REGION Network 108: M611-UNIT 02 FIXTURE 3 TWIN NC UNCLAMP SEQUENCE (TOGGLED) / M100-CLAMP SEQUENCE FIXTURE 1
   RUNG wire#powerrail
      Contact( "DB334_EXTENDED_M_CODE_UNIT_02_STA_0".M_code[611] )
      wire#w1
      I_Contact( "DB334_EXTENDED_M_CODE_UNIT_02_STA_0".M_code[611] )
      wire#w2
      I_Contact( "DB356_M_UNIT_02_STA_0".M_CODES_UNIT_02_STA_0.Ack_M611 )
      I_Contact( "DB2120_MPP_ITC_IPC".RESET_FAULTS )
      I_Contact( "DB356_M_UNIT_02_STA_0".M_CODES_UNIT_02_STA_0.M_RESET_PULSE )
      Coil( "DB356_M_UNIT_02_STA_0".M_CODES_UNIT_02_STA_0.M611 )
   END_RUNG
   RUNG wire#powerrail
      Contact( "DB356_M_UNIT_02_STA_0".M_CODES_UNIT_02_STA_0.M611 )
   END_RUNG wire#w1
   RUNG wire#w1
      I_Contact( "DB356_M_UNIT_02_STA_0".M_CODES_UNIT_02_STA_0.M611 )
   END_RUNG wire#w2
   // the same network as SCL:
   "DB356_M_UNIT_02_STA_0".M_CODES_UNIT_02_STA_0.M611 := ("DB334_EXTENDED_M_CODE_UNIT_02_STA_0".M_code[611] OR "DB356_M_UNIT_02_STA_0".M_CODES_UNIT_02_STA_0.M611) AND (NOT "DB334_EXTENDED_M_CODE_UNIT_02_STA_0".M_code[611] OR NOT "DB356_M_UNIT_02_STA_0".M_CODES_UNIT_02_STA_0.M611) AND NOT "DB356_M_UNIT_02_STA_0".M_CODES_UNIT_02_STA_0.Ack_M611 AND NOT "DB2120_MPP_ITC_IPC".RESET_FAULTS AND NOT "DB356_M_UNIT_02_STA_0".M_CODES_UNIT_02_STA_0.M_RESET_PULSE;
END_REGION

REGION Network 109: ACKNOWLEDGE M620- UNIT 02 FIXTURE 3 GRIPPER CLOSE (READ-IN DISABLE)
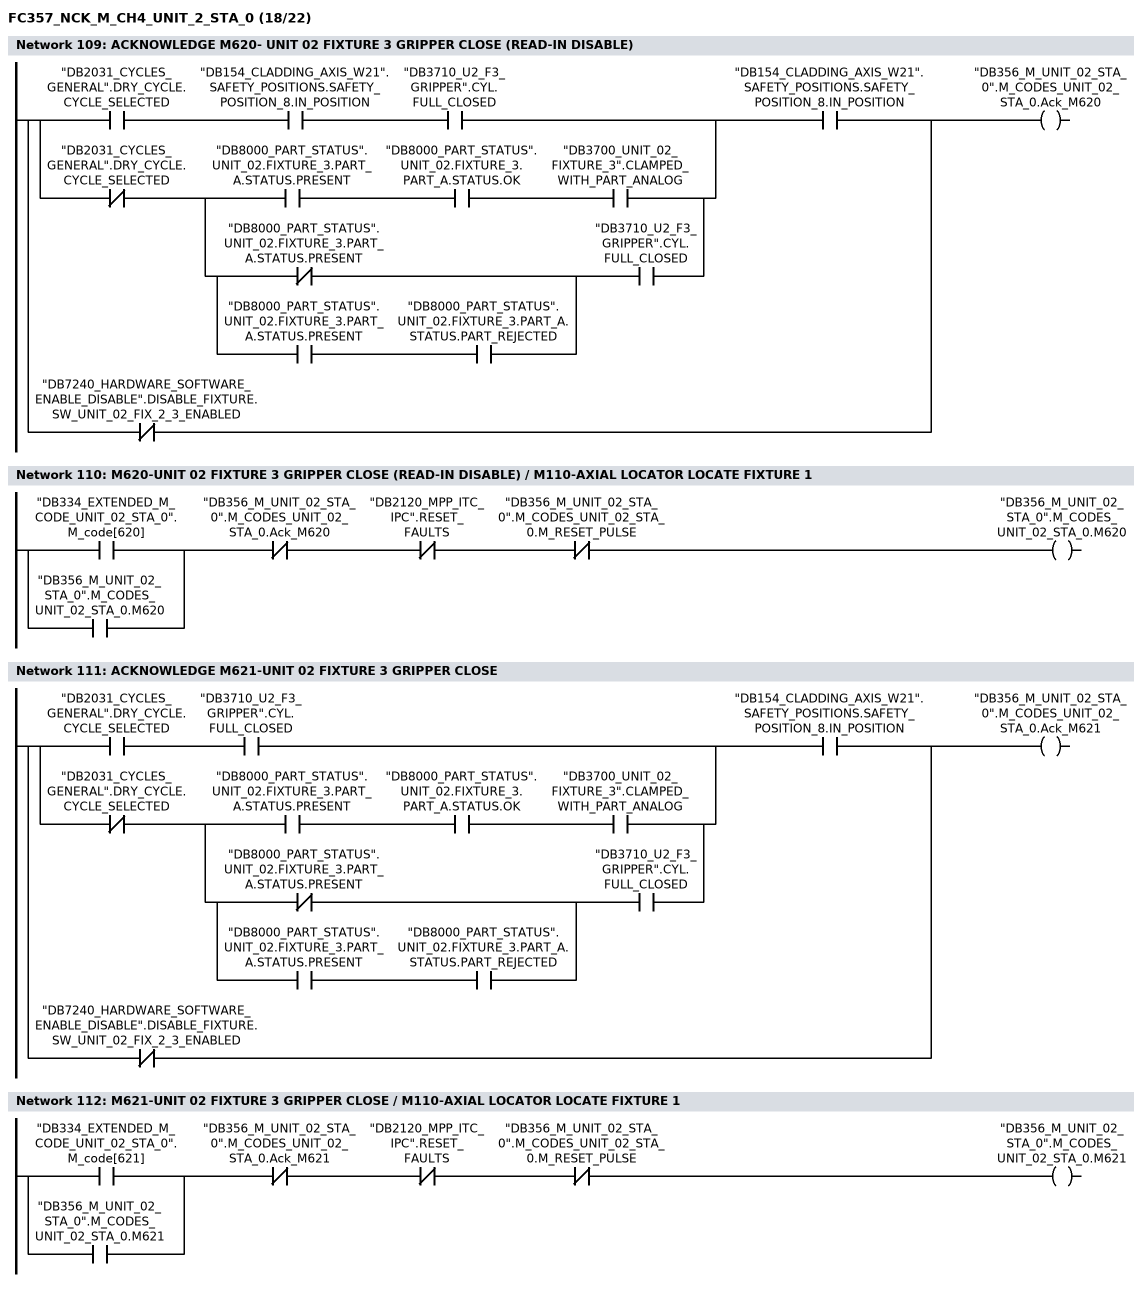
   RUNG wire#powerrail
      Contact( "DB2031_CYCLES_GENERAL".DRY_CYCLE.CYCLE_SELECTED )
      Contact( "DB154_CLADDING_AXIS_W21".SAFETY_POSITIONS.SAFETY_POSITION_8.IN_POSITION )
      Contact( "DB3710_U2_F3_GRIPPER".CYL.FULL_CLOSED )
      wire#w1
      Contact( "DB154_CLADDING_AXIS_W21".SAFETY_POSITIONS.SAFETY_POSITION_8.IN_POSITION )
      wire#w4
      Coil( "DB356_M_UNIT_02_STA_0".M_CODES_UNIT_02_STA_0.Ack_M620 )
   END_RUNG
   RUNG wire#powerrail
      I_Contact( "DB2031_CYCLES_GENERAL".DRY_CYCLE.CYCLE_SELECTED )
      wire#w2
      Contact( "DB8000_PART_STATUS".UNIT_02.FIXTURE_3.PART_A.STATUS.PRESENT )
      Contact( "DB8000_PART_STATUS".UNIT_02.FIXTURE_3.PART_A.STATUS.OK )
      Contact( "DB3700_UNIT_02_FIXTURE_3".CLAMPED_WITH_PART_ANALOG )
   END_RUNG wire#w1
   RUNG wire#w2
      I_Contact( "DB8000_PART_STATUS".UNIT_02.FIXTURE_3.PART_A.STATUS.PRESENT )
      wire#w3
      Contact( "DB3710_U2_F3_GRIPPER".CYL.FULL_CLOSED )
   END_RUNG wire#w1
   RUNG wire#w2
      Contact( "DB8000_PART_STATUS".UNIT_02.FIXTURE_3.PART_A.STATUS.PRESENT )
      Contact( "DB8000_PART_STATUS".UNIT_02.FIXTURE_3.PART_A.STATUS.PART_REJECTED )
   END_RUNG wire#w3
   RUNG wire#powerrail
      I_Contact( "DB7240_HARDWARE_SOFTWARE_ENABLE_DISABLE".DISABLE_FIXTURE.SW_UNIT_02_FIX_2_3_ENABLED )
   END_RUNG wire#w4
   // the same network as SCL:
   "DB356_M_UNIT_02_STA_0".M_CODES_UNIT_02_STA_0.Ack_M620 := ((("DB2031_CYCLES_GENERAL".DRY_CYCLE.CYCLE_SELECTED AND "DB154_CLADDING_AXIS_W21".SAFETY_POSITIONS.SAFETY_POSITION_8.IN_POSITION AND "DB3710_U2_F3_GRIPPER".CYL.FULL_CLOSED) OR (NOT "DB2031_CYCLES_GENERAL".DRY_CYCLE.CYCLE_SELECTED AND (("DB8000_PART_STATUS".UNIT_02.FIXTURE_3.PART_A.STATUS.PRESENT AND "DB8000_PART_STATUS".UNIT_02.FIXTURE_3.PART_A.STATUS.OK AND "DB3700_UNIT_02_FIXTURE_3".CLAMPED_WITH_PART_ANALOG) OR ((NOT "DB8000_PART_STATUS".UNIT_02.FIXTURE_3.PART_A.STATUS.PRESENT OR ("DB8000_PART_STATUS".UNIT_02.FIXTURE_3.PART_A.STATUS.PRESENT AND "DB8000_PART_STATUS".UNIT_02.FIXTURE_3.PART_A.STATUS.PART_REJECTED)) AND "DB3710_U2_F3_GRIPPER".CYL.FULL_CLOSED)))) AND "DB154_CLADDING_AXIS_W21".SAFETY_POSITIONS.SAFETY_POSITION_8.IN_POSITION) OR NOT "DB7240_HARDWARE_SOFTWARE_ENABLE_DISABLE".DISABLE_FIXTURE.SW_UNIT_02_FIX_2_3_ENABLED;
END_REGION

REGION Network 110: M620-UNIT 02 FIXTURE 3 GRIPPER CLOSE (READ-IN DISABLE) / M110-AXIAL LOCATOR LOCATE FIXTURE 1
   RUNG wire#powerrail
      Contact( "DB334_EXTENDED_M_CODE_UNIT_02_STA_0".M_code[620] )
      wire#w1
      I_Contact( "DB356_M_UNIT_02_STA_0".M_CODES_UNIT_02_STA_0.Ack_M620 )
      I_Contact( "DB2120_MPP_ITC_IPC".RESET_FAULTS )
      I_Contact( "DB356_M_UNIT_02_STA_0".M_CODES_UNIT_02_STA_0.M_RESET_PULSE )
      Coil( "DB356_M_UNIT_02_STA_0".M_CODES_UNIT_02_STA_0.M620 )
   END_RUNG
   RUNG wire#powerrail
      Contact( "DB356_M_UNIT_02_STA_0".M_CODES_UNIT_02_STA_0.M620 )
   END_RUNG wire#w1
   // the same network as SCL:
   "DB356_M_UNIT_02_STA_0".M_CODES_UNIT_02_STA_0.M620 := ("DB334_EXTENDED_M_CODE_UNIT_02_STA_0".M_code[620] OR "DB356_M_UNIT_02_STA_0".M_CODES_UNIT_02_STA_0.M620) AND NOT "DB356_M_UNIT_02_STA_0".M_CODES_UNIT_02_STA_0.Ack_M620 AND NOT "DB2120_MPP_ITC_IPC".RESET_FAULTS AND NOT "DB356_M_UNIT_02_STA_0".M_CODES_UNIT_02_STA_0.M_RESET_PULSE;
END_REGION

REGION Network 111: ACKNOWLEDGE M621-UNIT 02 FIXTURE 3 GRIPPER CLOSE
   RUNG wire#powerrail
      Contact( "DB2031_CYCLES_GENERAL".DRY_CYCLE.CYCLE_SELECTED )
      Contact( "DB3710_U2_F3_GRIPPER".CYL.FULL_CLOSED )
      wire#w1
      Contact( "DB154_CLADDING_AXIS_W21".SAFETY_POSITIONS.SAFETY_POSITION_8.IN_POSITION )
      wire#w4
      Coil( "DB356_M_UNIT_02_STA_0".M_CODES_UNIT_02_STA_0.Ack_M621 )
   END_RUNG
   RUNG wire#powerrail
      I_Contact( "DB2031_CYCLES_GENERAL".DRY_CYCLE.CYCLE_SELECTED )
      wire#w2
      Contact( "DB8000_PART_STATUS".UNIT_02.FIXTURE_3.PART_A.STATUS.PRESENT )
      Contact( "DB8000_PART_STATUS".UNIT_02.FIXTURE_3.PART_A.STATUS.OK )
      Contact( "DB3700_UNIT_02_FIXTURE_3".CLAMPED_WITH_PART_ANALOG )
   END_RUNG wire#w1
   RUNG wire#w2
      I_Contact( "DB8000_PART_STATUS".UNIT_02.FIXTURE_3.PART_A.STATUS.PRESENT )
      wire#w3
      Contact( "DB3710_U2_F3_GRIPPER".CYL.FULL_CLOSED )
   END_RUNG wire#w1
   RUNG wire#w2
      Contact( "DB8000_PART_STATUS".UNIT_02.FIXTURE_3.PART_A.STATUS.PRESENT )
      Contact( "DB8000_PART_STATUS".UNIT_02.FIXTURE_3.PART_A.STATUS.PART_REJECTED )
   END_RUNG wire#w3
   RUNG wire#powerrail
      I_Contact( "DB7240_HARDWARE_SOFTWARE_ENABLE_DISABLE".DISABLE_FIXTURE.SW_UNIT_02_FIX_2_3_ENABLED )
   END_RUNG wire#w4
   // the same network as SCL:
   "DB356_M_UNIT_02_STA_0".M_CODES_UNIT_02_STA_0.Ack_M621 := ((("DB2031_CYCLES_GENERAL".DRY_CYCLE.CYCLE_SELECTED AND "DB3710_U2_F3_GRIPPER".CYL.FULL_CLOSED) OR (NOT "DB2031_CYCLES_GENERAL".DRY_CYCLE.CYCLE_SELECTED AND (("DB8000_PART_STATUS".UNIT_02.FIXTURE_3.PART_A.STATUS.PRESENT AND "DB8000_PART_STATUS".UNIT_02.FIXTURE_3.PART_A.STATUS.OK AND "DB3700_UNIT_02_FIXTURE_3".CLAMPED_WITH_PART_ANALOG) OR ((NOT "DB8000_PART_STATUS".UNIT_02.FIXTURE_3.PART_A.STATUS.PRESENT OR ("DB8000_PART_STATUS".UNIT_02.FIXTURE_3.PART_A.STATUS.PRESENT AND "DB8000_PART_STATUS".UNIT_02.FIXTURE_3.PART_A.STATUS.PART_REJECTED)) AND "DB3710_U2_F3_GRIPPER".CYL.FULL_CLOSED)))) AND "DB154_CLADDING_AXIS_W21".SAFETY_POSITIONS.SAFETY_POSITION_8.IN_POSITION) OR NOT "DB7240_HARDWARE_SOFTWARE_ENABLE_DISABLE".DISABLE_FIXTURE.SW_UNIT_02_FIX_2_3_ENABLED;
END_REGION

REGION Network 112: M621-UNIT 02 FIXTURE 3 GRIPPER CLOSE / M110-AXIAL LOCATOR LOCATE FIXTURE 1
   RUNG wire#powerrail
      Contact( "DB334_EXTENDED_M_CODE_UNIT_02_STA_0".M_code[621] )
      wire#w1
      I_Contact( "DB356_M_UNIT_02_STA_0".M_CODES_UNIT_02_STA_0.Ack_M621 )
      I_Contact( "DB2120_MPP_ITC_IPC".RESET_FAULTS )
      I_Contact( "DB356_M_UNIT_02_STA_0".M_CODES_UNIT_02_STA_0.M_RESET_PULSE )
      Coil( "DB356_M_UNIT_02_STA_0".M_CODES_UNIT_02_STA_0.M621 )
   END_RUNG
   RUNG wire#powerrail
      Contact( "DB356_M_UNIT_02_STA_0".M_CODES_UNIT_02_STA_0.M621 )
   END_RUNG wire#w1
   // the same network as SCL:
   "DB356_M_UNIT_02_STA_0".M_CODES_UNIT_02_STA_0.M621 := ("DB334_EXTENDED_M_CODE_UNIT_02_STA_0".M_code[621] OR "DB356_M_UNIT_02_STA_0".M_CODES_UNIT_02_STA_0.M621) AND NOT "DB356_M_UNIT_02_STA_0".M_CODES_UNIT_02_STA_0.Ack_M621 AND NOT "DB2120_MPP_ITC_IPC".RESET_FAULTS AND NOT "DB356_M_UNIT_02_STA_0".M_CODES_UNIT_02_STA_0.M_RESET_PULSE;
END_REGION

REGION Network 113: ACKNOWLEDGE M622-UNIT 02 FIXTURE 3 GRIPPER OPEN (READ-IN DISABLE) / ACKNOWLEDGE M111-AXIAL LOCATOR RETURN FIXTURE 1
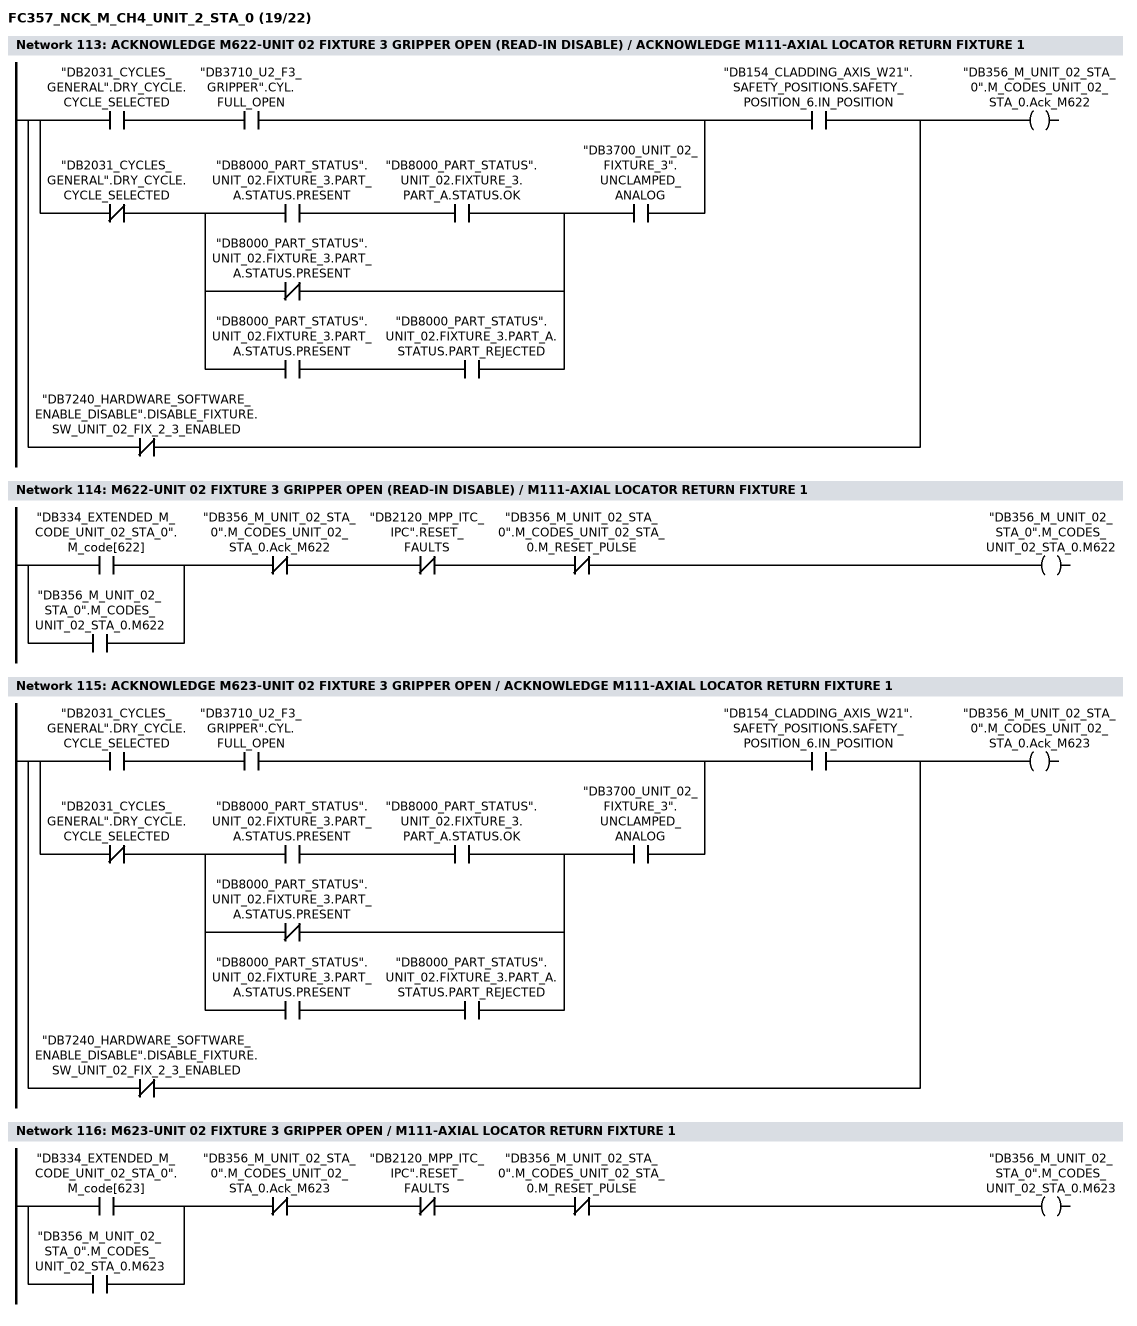
   RUNG wire#powerrail
      Contact( "DB2031_CYCLES_GENERAL".DRY_CYCLE.CYCLE_SELECTED )
      Contact( "DB3710_U2_F3_GRIPPER".CYL.FULL_OPEN )
      wire#w1
      Contact( "DB154_CLADDING_AXIS_W21".SAFETY_POSITIONS.SAFETY_POSITION_6.IN_POSITION )
      wire#w4
      Coil( "DB356_M_UNIT_02_STA_0".M_CODES_UNIT_02_STA_0.Ack_M622 )
   END_RUNG
   RUNG wire#powerrail
      I_Contact( "DB2031_CYCLES_GENERAL".DRY_CYCLE.CYCLE_SELECTED )
      wire#w2
      Contact( "DB8000_PART_STATUS".UNIT_02.FIXTURE_3.PART_A.STATUS.PRESENT )
      Contact( "DB8000_PART_STATUS".UNIT_02.FIXTURE_3.PART_A.STATUS.OK )
      wire#w3
      Contact( "DB3700_UNIT_02_FIXTURE_3".UNCLAMPED_ANALOG )
   END_RUNG wire#w1
   RUNG wire#w2
      I_Contact( "DB8000_PART_STATUS".UNIT_02.FIXTURE_3.PART_A.STATUS.PRESENT )
   END_RUNG wire#w3
   RUNG wire#w2
      Contact( "DB8000_PART_STATUS".UNIT_02.FIXTURE_3.PART_A.STATUS.PRESENT )
      Contact( "DB8000_PART_STATUS".UNIT_02.FIXTURE_3.PART_A.STATUS.PART_REJECTED )
   END_RUNG wire#w3
   RUNG wire#powerrail
      I_Contact( "DB7240_HARDWARE_SOFTWARE_ENABLE_DISABLE".DISABLE_FIXTURE.SW_UNIT_02_FIX_2_3_ENABLED )
   END_RUNG wire#w4
   // the same network as SCL:
   "DB356_M_UNIT_02_STA_0".M_CODES_UNIT_02_STA_0.Ack_M622 := ((("DB2031_CYCLES_GENERAL".DRY_CYCLE.CYCLE_SELECTED AND "DB3710_U2_F3_GRIPPER".CYL.FULL_OPEN) OR (NOT "DB2031_CYCLES_GENERAL".DRY_CYCLE.CYCLE_SELECTED AND (("DB8000_PART_STATUS".UNIT_02.FIXTURE_3.PART_A.STATUS.PRESENT AND "DB8000_PART_STATUS".UNIT_02.FIXTURE_3.PART_A.STATUS.OK) OR NOT "DB8000_PART_STATUS".UNIT_02.FIXTURE_3.PART_A.STATUS.PRESENT OR ("DB8000_PART_STATUS".UNIT_02.FIXTURE_3.PART_A.STATUS.PRESENT AND "DB8000_PART_STATUS".UNIT_02.FIXTURE_3.PART_A.STATUS.PART_REJECTED)) AND "DB3700_UNIT_02_FIXTURE_3".UNCLAMPED_ANALOG)) AND "DB154_CLADDING_AXIS_W21".SAFETY_POSITIONS.SAFETY_POSITION_6.IN_POSITION) OR NOT "DB7240_HARDWARE_SOFTWARE_ENABLE_DISABLE".DISABLE_FIXTURE.SW_UNIT_02_FIX_2_3_ENABLED;
END_REGION

REGION Network 114: M622-UNIT 02 FIXTURE 3 GRIPPER OPEN (READ-IN DISABLE) / M111-AXIAL LOCATOR RETURN FIXTURE 1
   RUNG wire#powerrail
      Contact( "DB334_EXTENDED_M_CODE_UNIT_02_STA_0".M_code[622] )
      wire#w1
      I_Contact( "DB356_M_UNIT_02_STA_0".M_CODES_UNIT_02_STA_0.Ack_M622 )
      I_Contact( "DB2120_MPP_ITC_IPC".RESET_FAULTS )
      I_Contact( "DB356_M_UNIT_02_STA_0".M_CODES_UNIT_02_STA_0.M_RESET_PULSE )
      Coil( "DB356_M_UNIT_02_STA_0".M_CODES_UNIT_02_STA_0.M622 )
   END_RUNG
   RUNG wire#powerrail
      Contact( "DB356_M_UNIT_02_STA_0".M_CODES_UNIT_02_STA_0.M622 )
   END_RUNG wire#w1
   // the same network as SCL:
   "DB356_M_UNIT_02_STA_0".M_CODES_UNIT_02_STA_0.M622 := ("DB334_EXTENDED_M_CODE_UNIT_02_STA_0".M_code[622] OR "DB356_M_UNIT_02_STA_0".M_CODES_UNIT_02_STA_0.M622) AND NOT "DB356_M_UNIT_02_STA_0".M_CODES_UNIT_02_STA_0.Ack_M622 AND NOT "DB2120_MPP_ITC_IPC".RESET_FAULTS AND NOT "DB356_M_UNIT_02_STA_0".M_CODES_UNIT_02_STA_0.M_RESET_PULSE;
END_REGION

REGION Network 115: ACKNOWLEDGE M623-UNIT 02 FIXTURE 3 GRIPPER OPEN / ACKNOWLEDGE M111-AXIAL LOCATOR RETURN FIXTURE 1
   RUNG wire#powerrail
      Contact( "DB2031_CYCLES_GENERAL".DRY_CYCLE.CYCLE_SELECTED )
      Contact( "DB3710_U2_F3_GRIPPER".CYL.FULL_OPEN )
      wire#w1
      Contact( "DB154_CLADDING_AXIS_W21".SAFETY_POSITIONS.SAFETY_POSITION_6.IN_POSITION )
      wire#w4
      Coil( "DB356_M_UNIT_02_STA_0".M_CODES_UNIT_02_STA_0.Ack_M623 )
   END_RUNG
   RUNG wire#powerrail
      I_Contact( "DB2031_CYCLES_GENERAL".DRY_CYCLE.CYCLE_SELECTED )
      wire#w2
      Contact( "DB8000_PART_STATUS".UNIT_02.FIXTURE_3.PART_A.STATUS.PRESENT )
      Contact( "DB8000_PART_STATUS".UNIT_02.FIXTURE_3.PART_A.STATUS.OK )
      wire#w3
      Contact( "DB3700_UNIT_02_FIXTURE_3".UNCLAMPED_ANALOG )
   END_RUNG wire#w1
   RUNG wire#w2
      I_Contact( "DB8000_PART_STATUS".UNIT_02.FIXTURE_3.PART_A.STATUS.PRESENT )
   END_RUNG wire#w3
   RUNG wire#w2
      Contact( "DB8000_PART_STATUS".UNIT_02.FIXTURE_3.PART_A.STATUS.PRESENT )
      Contact( "DB8000_PART_STATUS".UNIT_02.FIXTURE_3.PART_A.STATUS.PART_REJECTED )
   END_RUNG wire#w3
   RUNG wire#powerrail
      I_Contact( "DB7240_HARDWARE_SOFTWARE_ENABLE_DISABLE".DISABLE_FIXTURE.SW_UNIT_02_FIX_2_3_ENABLED )
   END_RUNG wire#w4
   // the same network as SCL:
   "DB356_M_UNIT_02_STA_0".M_CODES_UNIT_02_STA_0.Ack_M623 := ((("DB2031_CYCLES_GENERAL".DRY_CYCLE.CYCLE_SELECTED AND "DB3710_U2_F3_GRIPPER".CYL.FULL_OPEN) OR (NOT "DB2031_CYCLES_GENERAL".DRY_CYCLE.CYCLE_SELECTED AND (("DB8000_PART_STATUS".UNIT_02.FIXTURE_3.PART_A.STATUS.PRESENT AND "DB8000_PART_STATUS".UNIT_02.FIXTURE_3.PART_A.STATUS.OK) OR NOT "DB8000_PART_STATUS".UNIT_02.FIXTURE_3.PART_A.STATUS.PRESENT OR ("DB8000_PART_STATUS".UNIT_02.FIXTURE_3.PART_A.STATUS.PRESENT AND "DB8000_PART_STATUS".UNIT_02.FIXTURE_3.PART_A.STATUS.PART_REJECTED)) AND "DB3700_UNIT_02_FIXTURE_3".UNCLAMPED_ANALOG)) AND "DB154_CLADDING_AXIS_W21".SAFETY_POSITIONS.SAFETY_POSITION_6.IN_POSITION) OR NOT "DB7240_HARDWARE_SOFTWARE_ENABLE_DISABLE".DISABLE_FIXTURE.SW_UNIT_02_FIX_2_3_ENABLED;
END_REGION

REGION Network 116: M623-UNIT 02 FIXTURE 3 GRIPPER OPEN / M111-AXIAL LOCATOR RETURN FIXTURE 1
   RUNG wire#powerrail
      Contact( "DB334_EXTENDED_M_CODE_UNIT_02_STA_0".M_code[623] )
      wire#w1
      I_Contact( "DB356_M_UNIT_02_STA_0".M_CODES_UNIT_02_STA_0.Ack_M623 )
      I_Contact( "DB2120_MPP_ITC_IPC".RESET_FAULTS )
      I_Contact( "DB356_M_UNIT_02_STA_0".M_CODES_UNIT_02_STA_0.M_RESET_PULSE )
      Coil( "DB356_M_UNIT_02_STA_0".M_CODES_UNIT_02_STA_0.M623 )
   END_RUNG
   RUNG wire#powerrail
      Contact( "DB356_M_UNIT_02_STA_0".M_CODES_UNIT_02_STA_0.M623 )
   END_RUNG wire#w1
   // the same network as SCL:
   "DB356_M_UNIT_02_STA_0".M_CODES_UNIT_02_STA_0.M623 := ("DB334_EXTENDED_M_CODE_UNIT_02_STA_0".M_code[623] OR "DB356_M_UNIT_02_STA_0".M_CODES_UNIT_02_STA_0.M623) AND NOT "DB356_M_UNIT_02_STA_0".M_CODES_UNIT_02_STA_0.Ack_M623 AND NOT "DB2120_MPP_ITC_IPC".RESET_FAULTS AND NOT "DB356_M_UNIT_02_STA_0".M_CODES_UNIT_02_STA_0.M_RESET_PULSE;
END_REGION

REGION Network 117: ACKNOWLEDGE M624-UNIT 02 FIXTURE 3 GRIPPER RELEASE PRESSURE (READ-IN DISABLE) / ACKNOWLEDGE M112-AXIAL LOCATOR RELAX FIXTURE 1
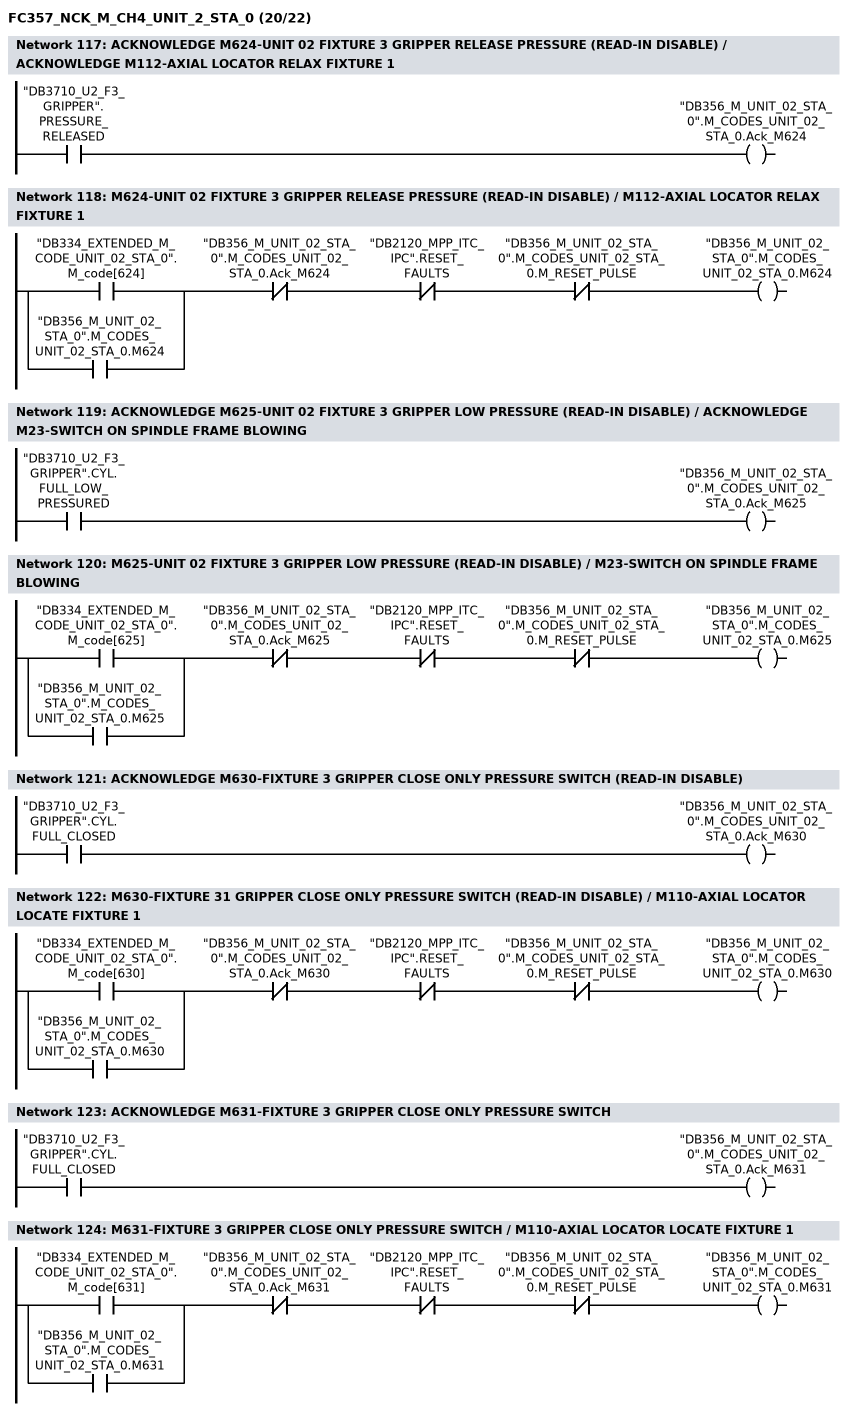
   RUNG wire#powerrail
      Contact( "DB3710_U2_F3_GRIPPER".PRESSURE_RELEASED )
      Coil( "DB356_M_UNIT_02_STA_0".M_CODES_UNIT_02_STA_0.Ack_M624 )
   END_RUNG
   // the same network as SCL:
   "DB356_M_UNIT_02_STA_0".M_CODES_UNIT_02_STA_0.Ack_M624 := "DB3710_U2_F3_GRIPPER".PRESSURE_RELEASED;
END_REGION

REGION Network 118: M624-UNIT 02 FIXTURE 3 GRIPPER RELEASE PRESSURE (READ-IN DISABLE) / M112-AXIAL LOCATOR RELAX FIXTURE 1
   RUNG wire#powerrail
      Contact( "DB334_EXTENDED_M_CODE_UNIT_02_STA_0".M_code[624] )
      wire#w1
      I_Contact( "DB356_M_UNIT_02_STA_0".M_CODES_UNIT_02_STA_0.Ack_M624 )
      I_Contact( "DB2120_MPP_ITC_IPC".RESET_FAULTS )
      I_Contact( "DB356_M_UNIT_02_STA_0".M_CODES_UNIT_02_STA_0.M_RESET_PULSE )
      Coil( "DB356_M_UNIT_02_STA_0".M_CODES_UNIT_02_STA_0.M624 )
   END_RUNG
   RUNG wire#powerrail
      Contact( "DB356_M_UNIT_02_STA_0".M_CODES_UNIT_02_STA_0.M624 )
   END_RUNG wire#w1
   // the same network as SCL:
   "DB356_M_UNIT_02_STA_0".M_CODES_UNIT_02_STA_0.M624 := ("DB334_EXTENDED_M_CODE_UNIT_02_STA_0".M_code[624] OR "DB356_M_UNIT_02_STA_0".M_CODES_UNIT_02_STA_0.M624) AND NOT "DB356_M_UNIT_02_STA_0".M_CODES_UNIT_02_STA_0.Ack_M624 AND NOT "DB2120_MPP_ITC_IPC".RESET_FAULTS AND NOT "DB356_M_UNIT_02_STA_0".M_CODES_UNIT_02_STA_0.M_RESET_PULSE;
END_REGION

REGION Network 119: ACKNOWLEDGE M625-UNIT 02 FIXTURE 3 GRIPPER LOW PRESSURE (READ-IN DISABLE) / ACKNOWLEDGE M23-SWITCH ON SPINDLE FRAME BLOWING
   RUNG wire#powerrail
      Contact( "DB3710_U2_F3_GRIPPER".CYL.FULL_LOW_PRESSURED )
      Coil( "DB356_M_UNIT_02_STA_0".M_CODES_UNIT_02_STA_0.Ack_M625 )
   END_RUNG
   // the same network as SCL:
   "DB356_M_UNIT_02_STA_0".M_CODES_UNIT_02_STA_0.Ack_M625 := "DB3710_U2_F3_GRIPPER".CYL.FULL_LOW_PRESSURED;
END_REGION

REGION Network 120: M625-UNIT 02 FIXTURE 3 GRIPPER LOW PRESSURE (READ-IN DISABLE) / M23-SWITCH ON SPINDLE FRAME BLOWING
   RUNG wire#powerrail
      Contact( "DB334_EXTENDED_M_CODE_UNIT_02_STA_0".M_code[625] )
      wire#w1
      I_Contact( "DB356_M_UNIT_02_STA_0".M_CODES_UNIT_02_STA_0.Ack_M625 )
      I_Contact( "DB2120_MPP_ITC_IPC".RESET_FAULTS )
      I_Contact( "DB356_M_UNIT_02_STA_0".M_CODES_UNIT_02_STA_0.M_RESET_PULSE )
      Coil( "DB356_M_UNIT_02_STA_0".M_CODES_UNIT_02_STA_0.M625 )
   END_RUNG
   RUNG wire#powerrail
      Contact( "DB356_M_UNIT_02_STA_0".M_CODES_UNIT_02_STA_0.M625 )
   END_RUNG wire#w1
   // the same network as SCL:
   "DB356_M_UNIT_02_STA_0".M_CODES_UNIT_02_STA_0.M625 := ("DB334_EXTENDED_M_CODE_UNIT_02_STA_0".M_code[625] OR "DB356_M_UNIT_02_STA_0".M_CODES_UNIT_02_STA_0.M625) AND NOT "DB356_M_UNIT_02_STA_0".M_CODES_UNIT_02_STA_0.Ack_M625 AND NOT "DB2120_MPP_ITC_IPC".RESET_FAULTS AND NOT "DB356_M_UNIT_02_STA_0".M_CODES_UNIT_02_STA_0.M_RESET_PULSE;
END_REGION

REGION Network 121: ACKNOWLEDGE M630-FIXTURE 3 GRIPPER CLOSE ONLY PRESSURE SWITCH (READ-IN DISABLE)
   RUNG wire#powerrail
      Contact( "DB3710_U2_F3_GRIPPER".CYL.FULL_CLOSED )
      Coil( "DB356_M_UNIT_02_STA_0".M_CODES_UNIT_02_STA_0.Ack_M630 )
   END_RUNG
   // the same network as SCL:
   "DB356_M_UNIT_02_STA_0".M_CODES_UNIT_02_STA_0.Ack_M630 := "DB3710_U2_F3_GRIPPER".CYL.FULL_CLOSED;
END_REGION

REGION Network 122: M630-FIXTURE 31 GRIPPER CLOSE ONLY PRESSURE SWITCH (READ-IN DISABLE) / M110-AXIAL LOCATOR LOCATE FIXTURE 1
   RUNG wire#powerrail
      Contact( "DB334_EXTENDED_M_CODE_UNIT_02_STA_0".M_code[630] )
      wire#w1
      I_Contact( "DB356_M_UNIT_02_STA_0".M_CODES_UNIT_02_STA_0.Ack_M630 )
      I_Contact( "DB2120_MPP_ITC_IPC".RESET_FAULTS )
      I_Contact( "DB356_M_UNIT_02_STA_0".M_CODES_UNIT_02_STA_0.M_RESET_PULSE )
      Coil( "DB356_M_UNIT_02_STA_0".M_CODES_UNIT_02_STA_0.M630 )
   END_RUNG
   RUNG wire#powerrail
      Contact( "DB356_M_UNIT_02_STA_0".M_CODES_UNIT_02_STA_0.M630 )
   END_RUNG wire#w1
   // the same network as SCL:
   "DB356_M_UNIT_02_STA_0".M_CODES_UNIT_02_STA_0.M630 := ("DB334_EXTENDED_M_CODE_UNIT_02_STA_0".M_code[630] OR "DB356_M_UNIT_02_STA_0".M_CODES_UNIT_02_STA_0.M630) AND NOT "DB356_M_UNIT_02_STA_0".M_CODES_UNIT_02_STA_0.Ack_M630 AND NOT "DB2120_MPP_ITC_IPC".RESET_FAULTS AND NOT "DB356_M_UNIT_02_STA_0".M_CODES_UNIT_02_STA_0.M_RESET_PULSE;
END_REGION

REGION Network 123: ACKNOWLEDGE M631-FIXTURE 3 GRIPPER CLOSE ONLY PRESSURE SWITCH
   RUNG wire#powerrail
      Contact( "DB3710_U2_F3_GRIPPER".CYL.FULL_CLOSED )
      Coil( "DB356_M_UNIT_02_STA_0".M_CODES_UNIT_02_STA_0.Ack_M631 )
   END_RUNG
   // the same network as SCL:
   "DB356_M_UNIT_02_STA_0".M_CODES_UNIT_02_STA_0.Ack_M631 := "DB3710_U2_F3_GRIPPER".CYL.FULL_CLOSED;
END_REGION

REGION Network 124: M631-FIXTURE 3 GRIPPER CLOSE ONLY PRESSURE SWITCH / M110-AXIAL LOCATOR LOCATE FIXTURE 1
   RUNG wire#powerrail
      Contact( "DB334_EXTENDED_M_CODE_UNIT_02_STA_0".M_code[631] )
      wire#w1
      I_Contact( "DB356_M_UNIT_02_STA_0".M_CODES_UNIT_02_STA_0.Ack_M631 )
      I_Contact( "DB2120_MPP_ITC_IPC".RESET_FAULTS )
      I_Contact( "DB356_M_UNIT_02_STA_0".M_CODES_UNIT_02_STA_0.M_RESET_PULSE )
      Coil( "DB356_M_UNIT_02_STA_0".M_CODES_UNIT_02_STA_0.M631 )
   END_RUNG
   RUNG wire#powerrail
      Contact( "DB356_M_UNIT_02_STA_0".M_CODES_UNIT_02_STA_0.M631 )
   END_RUNG wire#w1
   // the same network as SCL:
   "DB356_M_UNIT_02_STA_0".M_CODES_UNIT_02_STA_0.M631 := ("DB334_EXTENDED_M_CODE_UNIT_02_STA_0".M_code[631] OR "DB356_M_UNIT_02_STA_0".M_CODES_UNIT_02_STA_0.M631) AND NOT "DB356_M_UNIT_02_STA_0".M_CODES_UNIT_02_STA_0.Ack_M631 AND NOT "DB2120_MPP_ITC_IPC".RESET_FAULTS AND NOT "DB356_M_UNIT_02_STA_0".M_CODES_UNIT_02_STA_0.M_RESET_PULSE;
END_REGION

REGION Network 125: ACKNOWLEDGE M632-FIXTURE 3 GRIPPER OPEN ONLY PRESSURE SWITCH (READ-IN DISABLE) / ACKNOWLEDGE M111-AXIAL LOCATOR RETURN FIXTURE 1
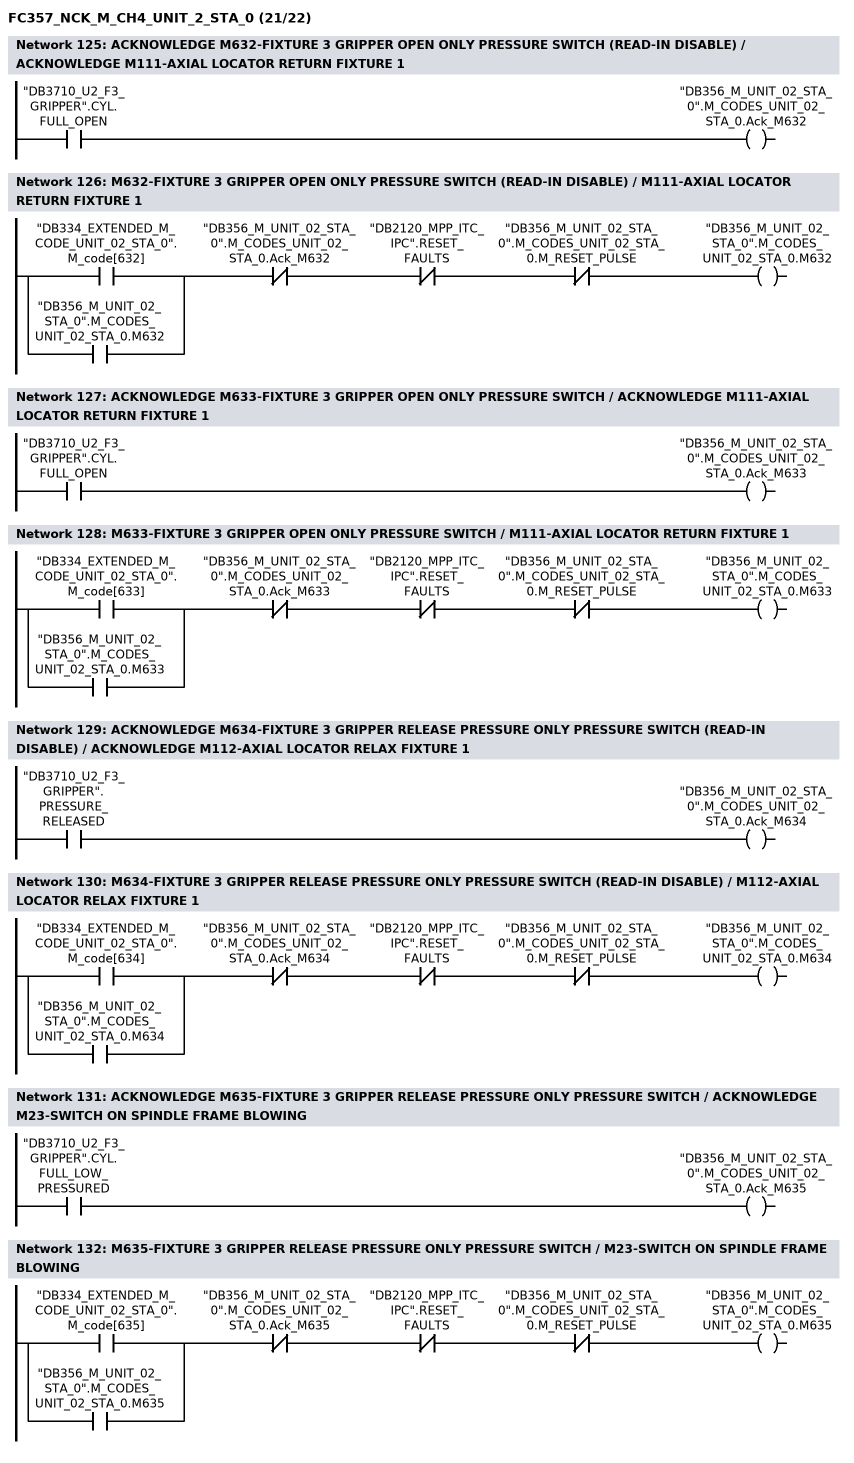
   RUNG wire#powerrail
      Contact( "DB3710_U2_F3_GRIPPER".CYL.FULL_OPEN )
      Coil( "DB356_M_UNIT_02_STA_0".M_CODES_UNIT_02_STA_0.Ack_M632 )
   END_RUNG
   // the same network as SCL:
   "DB356_M_UNIT_02_STA_0".M_CODES_UNIT_02_STA_0.Ack_M632 := "DB3710_U2_F3_GRIPPER".CYL.FULL_OPEN;
END_REGION

REGION Network 126: M632-FIXTURE 3 GRIPPER OPEN ONLY PRESSURE SWITCH (READ-IN DISABLE) / M111-AXIAL LOCATOR RETURN FIXTURE 1
   RUNG wire#powerrail
      Contact( "DB334_EXTENDED_M_CODE_UNIT_02_STA_0".M_code[632] )
      wire#w1
      I_Contact( "DB356_M_UNIT_02_STA_0".M_CODES_UNIT_02_STA_0.Ack_M632 )
      I_Contact( "DB2120_MPP_ITC_IPC".RESET_FAULTS )
      I_Contact( "DB356_M_UNIT_02_STA_0".M_CODES_UNIT_02_STA_0.M_RESET_PULSE )
      Coil( "DB356_M_UNIT_02_STA_0".M_CODES_UNIT_02_STA_0.M632 )
   END_RUNG
   RUNG wire#powerrail
      Contact( "DB356_M_UNIT_02_STA_0".M_CODES_UNIT_02_STA_0.M632 )
   END_RUNG wire#w1
   // the same network as SCL:
   "DB356_M_UNIT_02_STA_0".M_CODES_UNIT_02_STA_0.M632 := ("DB334_EXTENDED_M_CODE_UNIT_02_STA_0".M_code[632] OR "DB356_M_UNIT_02_STA_0".M_CODES_UNIT_02_STA_0.M632) AND NOT "DB356_M_UNIT_02_STA_0".M_CODES_UNIT_02_STA_0.Ack_M632 AND NOT "DB2120_MPP_ITC_IPC".RESET_FAULTS AND NOT "DB356_M_UNIT_02_STA_0".M_CODES_UNIT_02_STA_0.M_RESET_PULSE;
END_REGION

REGION Network 127: ACKNOWLEDGE M633-FIXTURE 3 GRIPPER OPEN ONLY PRESSURE SWITCH / ACKNOWLEDGE M111-AXIAL LOCATOR RETURN FIXTURE 1
   RUNG wire#powerrail
      Contact( "DB3710_U2_F3_GRIPPER".CYL.FULL_OPEN )
      Coil( "DB356_M_UNIT_02_STA_0".M_CODES_UNIT_02_STA_0.Ack_M633 )
   END_RUNG
   // the same network as SCL:
   "DB356_M_UNIT_02_STA_0".M_CODES_UNIT_02_STA_0.Ack_M633 := "DB3710_U2_F3_GRIPPER".CYL.FULL_OPEN;
END_REGION

REGION Network 128: M633-FIXTURE 3 GRIPPER OPEN ONLY PRESSURE SWITCH / M111-AXIAL LOCATOR RETURN FIXTURE 1
   RUNG wire#powerrail
      Contact( "DB334_EXTENDED_M_CODE_UNIT_02_STA_0".M_code[633] )
      wire#w1
      I_Contact( "DB356_M_UNIT_02_STA_0".M_CODES_UNIT_02_STA_0.Ack_M633 )
      I_Contact( "DB2120_MPP_ITC_IPC".RESET_FAULTS )
      I_Contact( "DB356_M_UNIT_02_STA_0".M_CODES_UNIT_02_STA_0.M_RESET_PULSE )
      Coil( "DB356_M_UNIT_02_STA_0".M_CODES_UNIT_02_STA_0.M633 )
   END_RUNG
   RUNG wire#powerrail
      Contact( "DB356_M_UNIT_02_STA_0".M_CODES_UNIT_02_STA_0.M633 )
   END_RUNG wire#w1
   // the same network as SCL:
   "DB356_M_UNIT_02_STA_0".M_CODES_UNIT_02_STA_0.M633 := ("DB334_EXTENDED_M_CODE_UNIT_02_STA_0".M_code[633] OR "DB356_M_UNIT_02_STA_0".M_CODES_UNIT_02_STA_0.M633) AND NOT "DB356_M_UNIT_02_STA_0".M_CODES_UNIT_02_STA_0.Ack_M633 AND NOT "DB2120_MPP_ITC_IPC".RESET_FAULTS AND NOT "DB356_M_UNIT_02_STA_0".M_CODES_UNIT_02_STA_0.M_RESET_PULSE;
END_REGION

REGION Network 129: ACKNOWLEDGE M634-FIXTURE 3 GRIPPER RELEASE PRESSURE ONLY PRESSURE SWITCH (READ-IN DISABLE) / ACKNOWLEDGE M112-AXIAL LOCATOR RELAX FIXTURE 1
   RUNG wire#powerrail
      Contact( "DB3710_U2_F3_GRIPPER".PRESSURE_RELEASED )
      Coil( "DB356_M_UNIT_02_STA_0".M_CODES_UNIT_02_STA_0.Ack_M634 )
   END_RUNG
   // the same network as SCL:
   "DB356_M_UNIT_02_STA_0".M_CODES_UNIT_02_STA_0.Ack_M634 := "DB3710_U2_F3_GRIPPER".PRESSURE_RELEASED;
END_REGION

REGION Network 130: M634-FIXTURE 3 GRIPPER RELEASE PRESSURE ONLY PRESSURE SWITCH (READ-IN DISABLE) / M112-AXIAL LOCATOR RELAX FIXTURE 1
   RUNG wire#powerrail
      Contact( "DB334_EXTENDED_M_CODE_UNIT_02_STA_0".M_code[634] )
      wire#w1
      I_Contact( "DB356_M_UNIT_02_STA_0".M_CODES_UNIT_02_STA_0.Ack_M634 )
      I_Contact( "DB2120_MPP_ITC_IPC".RESET_FAULTS )
      I_Contact( "DB356_M_UNIT_02_STA_0".M_CODES_UNIT_02_STA_0.M_RESET_PULSE )
      Coil( "DB356_M_UNIT_02_STA_0".M_CODES_UNIT_02_STA_0.M634 )
   END_RUNG
   RUNG wire#powerrail
      Contact( "DB356_M_UNIT_02_STA_0".M_CODES_UNIT_02_STA_0.M634 )
   END_RUNG wire#w1
   // the same network as SCL:
   "DB356_M_UNIT_02_STA_0".M_CODES_UNIT_02_STA_0.M634 := ("DB334_EXTENDED_M_CODE_UNIT_02_STA_0".M_code[634] OR "DB356_M_UNIT_02_STA_0".M_CODES_UNIT_02_STA_0.M634) AND NOT "DB356_M_UNIT_02_STA_0".M_CODES_UNIT_02_STA_0.Ack_M634 AND NOT "DB2120_MPP_ITC_IPC".RESET_FAULTS AND NOT "DB356_M_UNIT_02_STA_0".M_CODES_UNIT_02_STA_0.M_RESET_PULSE;
END_REGION

REGION Network 131: ACKNOWLEDGE M635-FIXTURE 3 GRIPPER RELEASE PRESSURE ONLY PRESSURE SWITCH / ACKNOWLEDGE M23-SWITCH ON SPINDLE FRAME BLOWING
   RUNG wire#powerrail
      Contact( "DB3710_U2_F3_GRIPPER".CYL.FULL_LOW_PRESSURED )
      Coil( "DB356_M_UNIT_02_STA_0".M_CODES_UNIT_02_STA_0.Ack_M635 )
   END_RUNG
   // the same network as SCL:
   "DB356_M_UNIT_02_STA_0".M_CODES_UNIT_02_STA_0.Ack_M635 := "DB3710_U2_F3_GRIPPER".CYL.FULL_LOW_PRESSURED;
END_REGION

REGION Network 132: M635-FIXTURE 3 GRIPPER RELEASE PRESSURE ONLY PRESSURE SWITCH / M23-SWITCH ON SPINDLE FRAME BLOWING
   RUNG wire#powerrail
      Contact( "DB334_EXTENDED_M_CODE_UNIT_02_STA_0".M_code[635] )
      wire#w1
      I_Contact( "DB356_M_UNIT_02_STA_0".M_CODES_UNIT_02_STA_0.Ack_M635 )
      I_Contact( "DB2120_MPP_ITC_IPC".RESET_FAULTS )
      I_Contact( "DB356_M_UNIT_02_STA_0".M_CODES_UNIT_02_STA_0.M_RESET_PULSE )
      Coil( "DB356_M_UNIT_02_STA_0".M_CODES_UNIT_02_STA_0.M635 )
   END_RUNG
   RUNG wire#powerrail
      Contact( "DB356_M_UNIT_02_STA_0".M_CODES_UNIT_02_STA_0.M635 )
   END_RUNG wire#w1
   // the same network as SCL:
   "DB356_M_UNIT_02_STA_0".M_CODES_UNIT_02_STA_0.M635 := ("DB334_EXTENDED_M_CODE_UNIT_02_STA_0".M_code[635] OR "DB356_M_UNIT_02_STA_0".M_CODES_UNIT_02_STA_0.M635) AND NOT "DB356_M_UNIT_02_STA_0".M_CODES_UNIT_02_STA_0.Ack_M635 AND NOT "DB2120_MPP_ITC_IPC".RESET_FAULTS AND NOT "DB356_M_UNIT_02_STA_0".M_CODES_UNIT_02_STA_0.M_RESET_PULSE;
END_REGION

REGION Network 133: READ-IN DISABLE / Read-in disable
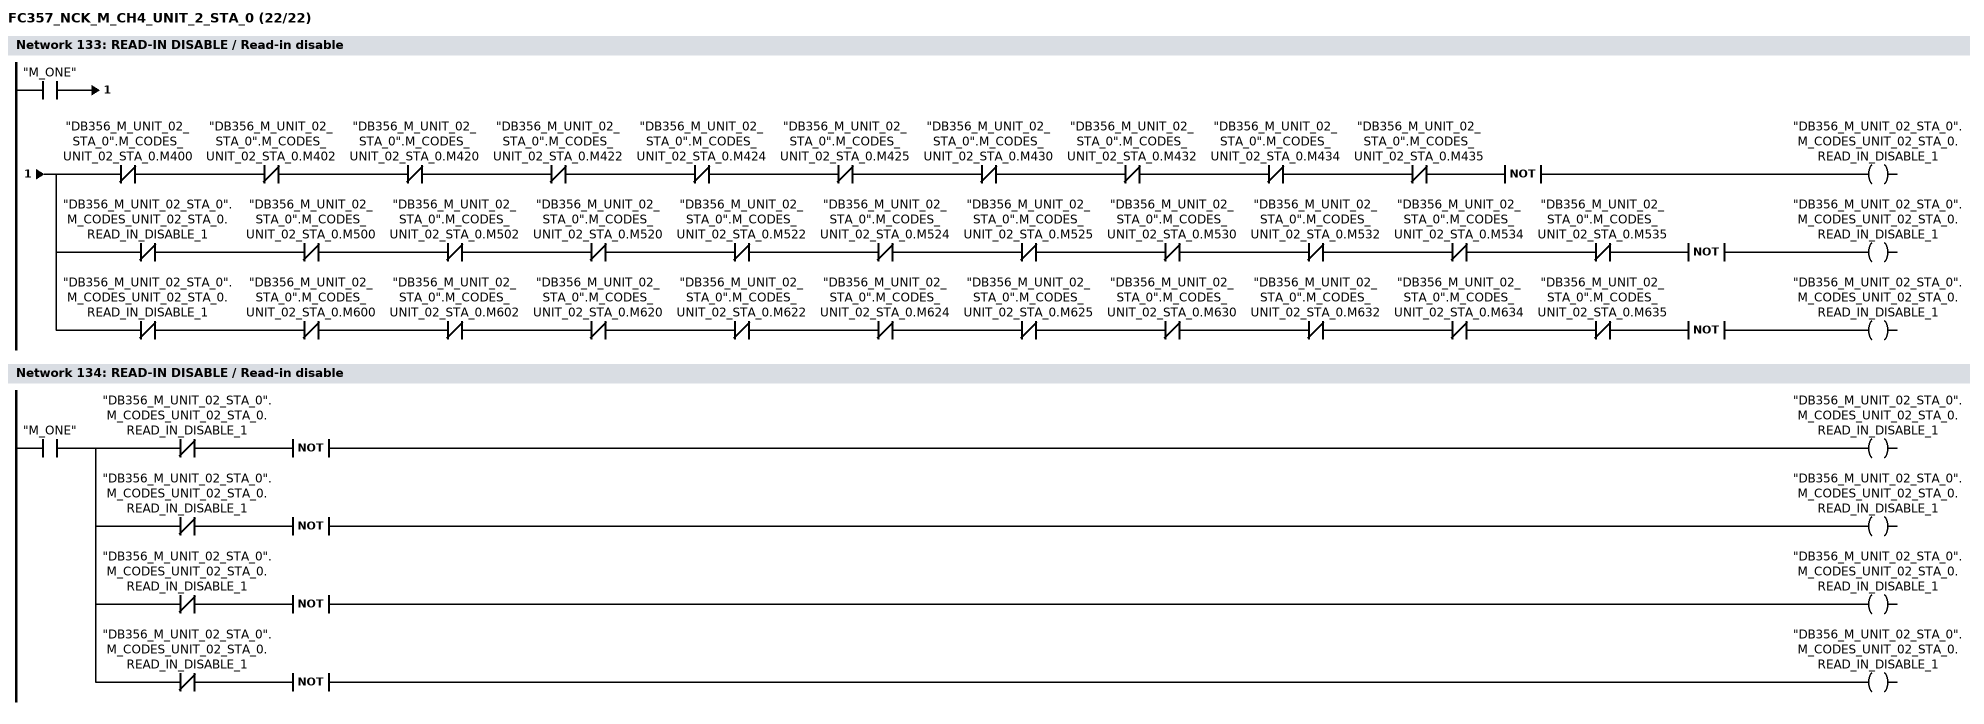
   RUNG wire#powerrail
      Contact( "M_ONE" )
      wire#w1
      I_Contact( "DB356_M_UNIT_02_STA_0".M_CODES_UNIT_02_STA_0.M400 )
      I_Contact( "DB356_M_UNIT_02_STA_0".M_CODES_UNIT_02_STA_0.M402 )
      I_Contact( "DB356_M_UNIT_02_STA_0".M_CODES_UNIT_02_STA_0.M420 )
      I_Contact( "DB356_M_UNIT_02_STA_0".M_CODES_UNIT_02_STA_0.M422 )
      I_Contact( "DB356_M_UNIT_02_STA_0".M_CODES_UNIT_02_STA_0.M424 )
      I_Contact( "DB356_M_UNIT_02_STA_0".M_CODES_UNIT_02_STA_0.M425 )
      I_Contact( "DB356_M_UNIT_02_STA_0".M_CODES_UNIT_02_STA_0.M430 )
      I_Contact( "DB356_M_UNIT_02_STA_0".M_CODES_UNIT_02_STA_0.M432 )
      I_Contact( "DB356_M_UNIT_02_STA_0".M_CODES_UNIT_02_STA_0.M434 )
      I_Contact( "DB356_M_UNIT_02_STA_0".M_CODES_UNIT_02_STA_0.M435 )
      Not()
      Coil( "DB356_M_UNIT_02_STA_0".M_CODES_UNIT_02_STA_0.READ_IN_DISABLE_1 )
   END_RUNG
   RUNG wire#w1
      I_Contact( "DB356_M_UNIT_02_STA_0".M_CODES_UNIT_02_STA_0.READ_IN_DISABLE_1 )
      I_Contact( "DB356_M_UNIT_02_STA_0".M_CODES_UNIT_02_STA_0.M500 )
      I_Contact( "DB356_M_UNIT_02_STA_0".M_CODES_UNIT_02_STA_0.M502 )
      I_Contact( "DB356_M_UNIT_02_STA_0".M_CODES_UNIT_02_STA_0.M520 )
      I_Contact( "DB356_M_UNIT_02_STA_0".M_CODES_UNIT_02_STA_0.M522 )
      I_Contact( "DB356_M_UNIT_02_STA_0".M_CODES_UNIT_02_STA_0.M524 )
      I_Contact( "DB356_M_UNIT_02_STA_0".M_CODES_UNIT_02_STA_0.M525 )
      I_Contact( "DB356_M_UNIT_02_STA_0".M_CODES_UNIT_02_STA_0.M530 )
      I_Contact( "DB356_M_UNIT_02_STA_0".M_CODES_UNIT_02_STA_0.M532 )
      I_Contact( "DB356_M_UNIT_02_STA_0".M_CODES_UNIT_02_STA_0.M534 )
      I_Contact( "DB356_M_UNIT_02_STA_0".M_CODES_UNIT_02_STA_0.M535 )
      Not()
      Coil( "DB356_M_UNIT_02_STA_0".M_CODES_UNIT_02_STA_0.READ_IN_DISABLE_1 )
   END_RUNG
   RUNG wire#w1
      I_Contact( "DB356_M_UNIT_02_STA_0".M_CODES_UNIT_02_STA_0.READ_IN_DISABLE_1 )
      I_Contact( "DB356_M_UNIT_02_STA_0".M_CODES_UNIT_02_STA_0.M600 )
      I_Contact( "DB356_M_UNIT_02_STA_0".M_CODES_UNIT_02_STA_0.M602 )
      I_Contact( "DB356_M_UNIT_02_STA_0".M_CODES_UNIT_02_STA_0.M620 )
      I_Contact( "DB356_M_UNIT_02_STA_0".M_CODES_UNIT_02_STA_0.M622 )
      I_Contact( "DB356_M_UNIT_02_STA_0".M_CODES_UNIT_02_STA_0.M624 )
      I_Contact( "DB356_M_UNIT_02_STA_0".M_CODES_UNIT_02_STA_0.M625 )
      I_Contact( "DB356_M_UNIT_02_STA_0".M_CODES_UNIT_02_STA_0.M630 )
      I_Contact( "DB356_M_UNIT_02_STA_0".M_CODES_UNIT_02_STA_0.M632 )
      I_Contact( "DB356_M_UNIT_02_STA_0".M_CODES_UNIT_02_STA_0.M634 )
      I_Contact( "DB356_M_UNIT_02_STA_0".M_CODES_UNIT_02_STA_0.M635 )
      Not()
      Coil( "DB356_M_UNIT_02_STA_0".M_CODES_UNIT_02_STA_0.READ_IN_DISABLE_1 )
   END_RUNG
   // the same network as SCL:
   "DB356_M_UNIT_02_STA_0".M_CODES_UNIT_02_STA_0.READ_IN_DISABLE_1 := NOT ("M_ONE" AND NOT "DB356_M_UNIT_02_STA_0".M_CODES_UNIT_02_STA_0.M400 AND NOT "DB356_M_UNIT_02_STA_0".M_CODES_UNIT_02_STA_0.M402 AND NOT "DB356_M_UNIT_02_STA_0".M_CODES_UNIT_02_STA_0.M420 AND NOT "DB356_M_UNIT_02_STA_0".M_CODES_UNIT_02_STA_0.M422 AND NOT "DB356_M_UNIT_02_STA_0".M_CODES_UNIT_02_STA_0.M424 AND NOT "DB356_M_UNIT_02_STA_0".M_CODES_UNIT_02_STA_0.M425 AND NOT "DB356_M_UNIT_02_STA_0".M_CODES_UNIT_02_STA_0.M430 AND NOT "DB356_M_UNIT_02_STA_0".M_CODES_UNIT_02_STA_0.M432 AND NOT "DB356_M_UNIT_02_STA_0".M_CODES_UNIT_02_STA_0.M434 AND NOT "DB356_M_UNIT_02_STA_0".M_CODES_UNIT_02_STA_0.M435);
   "DB356_M_UNIT_02_STA_0".M_CODES_UNIT_02_STA_0.READ_IN_DISABLE_1 := NOT ("M_ONE" AND NOT "DB356_M_UNIT_02_STA_0".M_CODES_UNIT_02_STA_0.READ_IN_DISABLE_1 AND NOT "DB356_M_UNIT_02_STA_0".M_CODES_UNIT_02_STA_0.M500 AND NOT "DB356_M_UNIT_02_STA_0".M_CODES_UNIT_02_STA_0.M502 AND NOT "DB356_M_UNIT_02_STA_0".M_CODES_UNIT_02_STA_0.M520 AND NOT "DB356_M_UNIT_02_STA_0".M_CODES_UNIT_02_STA_0.M522 AND NOT "DB356_M_UNIT_02_STA_0".M_CODES_UNIT_02_STA_0.M524 AND NOT "DB356_M_UNIT_02_STA_0".M_CODES_UNIT_02_STA_0.M525 AND NOT "DB356_M_UNIT_02_STA_0".M_CODES_UNIT_02_STA_0.M530 AND NOT "DB356_M_UNIT_02_STA_0".M_CODES_UNIT_02_STA_0.M532 AND NOT "DB356_M_UNIT_02_STA_0".M_CODES_UNIT_02_STA_0.M534 AND NOT "DB356_M_UNIT_02_STA_0".M_CODES_UNIT_02_STA_0.M535);
   "DB356_M_UNIT_02_STA_0".M_CODES_UNIT_02_STA_0.READ_IN_DISABLE_1 := NOT ("M_ONE" AND NOT "DB356_M_UNIT_02_STA_0".M_CODES_UNIT_02_STA_0.READ_IN_DISABLE_1 AND NOT "DB356_M_UNIT_02_STA_0".M_CODES_UNIT_02_STA_0.M600 AND NOT "DB356_M_UNIT_02_STA_0".M_CODES_UNIT_02_STA_0.M602 AND NOT "DB356_M_UNIT_02_STA_0".M_CODES_UNIT_02_STA_0.M620 AND NOT "DB356_M_UNIT_02_STA_0".M_CODES_UNIT_02_STA_0.M622 AND NOT "DB356_M_UNIT_02_STA_0".M_CODES_UNIT_02_STA_0.M624 AND NOT "DB356_M_UNIT_02_STA_0".M_CODES_UNIT_02_STA_0.M625 AND NOT "DB356_M_UNIT_02_STA_0".M_CODES_UNIT_02_STA_0.M630 AND NOT "DB356_M_UNIT_02_STA_0".M_CODES_UNIT_02_STA_0.M632 AND NOT "DB356_M_UNIT_02_STA_0".M_CODES_UNIT_02_STA_0.M634 AND NOT "DB356_M_UNIT_02_STA_0".M_CODES_UNIT_02_STA_0.M635);
END_REGION

REGION Network 134: READ-IN DISABLE / Read-in disable
   RUNG wire#powerrail
      Contact( "M_ONE" )
      wire#w1
      I_Contact( "DB356_M_UNIT_02_STA_0".M_CODES_UNIT_02_STA_0.READ_IN_DISABLE_1 )
      Not()
      Coil( "DB356_M_UNIT_02_STA_0".M_CODES_UNIT_02_STA_0.READ_IN_DISABLE_1 )
   END_RUNG
   RUNG wire#w1
      I_Contact( "DB356_M_UNIT_02_STA_0".M_CODES_UNIT_02_STA_0.READ_IN_DISABLE_1 )
      Not()
      Coil( "DB356_M_UNIT_02_STA_0".M_CODES_UNIT_02_STA_0.READ_IN_DISABLE_1 )
   END_RUNG
   RUNG wire#w1
      I_Contact( "DB356_M_UNIT_02_STA_0".M_CODES_UNIT_02_STA_0.READ_IN_DISABLE_1 )
      Not()
      Coil( "DB356_M_UNIT_02_STA_0".M_CODES_UNIT_02_STA_0.READ_IN_DISABLE_1 )
   END_RUNG
   RUNG wire#w1
      I_Contact( "DB356_M_UNIT_02_STA_0".M_CODES_UNIT_02_STA_0.READ_IN_DISABLE_1 )
      Not()
      Coil( "DB356_M_UNIT_02_STA_0".M_CODES_UNIT_02_STA_0.READ_IN_DISABLE_1 )
   END_RUNG
   // the same network as SCL:
   "DB356_M_UNIT_02_STA_0".M_CODES_UNIT_02_STA_0.READ_IN_DISABLE_1 := NOT ("M_ONE" AND NOT "DB356_M_UNIT_02_STA_0".M_CODES_UNIT_02_STA_0.READ_IN_DISABLE_1);
   "DB356_M_UNIT_02_STA_0".M_CODES_UNIT_02_STA_0.READ_IN_DISABLE_1 := NOT ("M_ONE" AND NOT "DB356_M_UNIT_02_STA_0".M_CODES_UNIT_02_STA_0.READ_IN_DISABLE_1);
   "DB356_M_UNIT_02_STA_0".M_CODES_UNIT_02_STA_0.READ_IN_DISABLE_1 := NOT ("M_ONE" AND NOT "DB356_M_UNIT_02_STA_0".M_CODES_UNIT_02_STA_0.READ_IN_DISABLE_1);
   "DB356_M_UNIT_02_STA_0".M_CODES_UNIT_02_STA_0.READ_IN_DISABLE_1 := NOT ("M_ONE" AND NOT "DB356_M_UNIT_02_STA_0".M_CODES_UNIT_02_STA_0.READ_IN_DISABLE_1);
END_REGION
END_FUNCTION
